// TIA Portal V19 export
DATA_BLOCK "iDBF_CaptiveKeyInLock"   // DB932, F_DB
{ DB_Accessible_From_OPC_UA := 'FALSE' }
// stored: AutoNumber false, DBAccessibleFromOPCUA false, DBAccessibleFromWebserver false, InstanceOfName EmergencyStop, InstanceOfType FB
"EmergencyStop"
   // VAR_INPUT
   //    xInputSafety { ExternalAccessible := 'False'; ExternalVisible := 'False'; ExternalWritable := 'False'} : Bool;
   //    xStateInput { ExternalAccessible := 'False'; ExternalVisible := 'False'; ExternalWritable := 'False'} : Bool;
   //    xAck { ExternalAccessible := 'False'; ExternalVisible := 'False'; ExternalWritable := 'False'} : Bool;
   //    xAllowAck { ExternalAccessible := 'False'; ExternalVisible := 'False'; ExternalWritable := 'False'} : Bool;
   // END_VAR
   // VAR_OUTPUT
   //    xStateSafety { ExternalAccessible := 'False'; ExternalVisible := 'False'; ExternalWritable := 'False'} : Bool;
   //    stSafetyState { ExternalAccessible := 'False'; ExternalVisible := 'False'; ExternalWritable := 'False'} : "stSafetyState";
   // END_VAR
   // VAR
   //    sx_Ack { ExternalAccessible := 'False'; ExternalVisible := 'False'; ExternalWritable := 'False'} : Bool;
   //    sx_TempAck { ExternalAccessible := 'False'; ExternalVisible := 'False'; ExternalWritable := 'False'} : Bool;
   //    sx_TempAckReq { ExternalAccessible := 'False'; ExternalVisible := 'False'; ExternalWritable := 'False'} : Bool;
   //    miDBF_EStop { ExternalAccessible := 'False'; ExternalVisible := 'False'; ExternalWritable := 'False'} : ESTOP1;
   // END_VAR
BEGIN
END_DATA_BLOCK
